TYPE TEngine :
STRUCT
	Cmd : TEngineCmd;
	State : TEngineState;
	Time2Start : TIME := T#5S;
	RisingEdgeTrigger : R_TRIG;
	StartupFailTimer : TON;
END_STRUCT
END_TYPE

(* stored: Version 1.1.0.1, ProductVersion 3.1.4024.12
   DUT TEngine: Id {b27109ba-b893-44c3-9a09-20e0a48b4f63} *)
